// TwinCAT 3 PLC project FB_RobotArm
// Company: DVKruglov
// ProjectVersion: 1.0
// ProgramVersion: 3.1.4023.0
// libraries:
//   Tc2_Standard, * (Beckhoff Automation GmbH)
//   Tc2_System, * (Beckhoff Automation GmbH)
//   Tc3_Module, * (Beckhoff Automation GmbH)
// project tree:
//   FB_RobotArmBase/Constants/ GVL_RobotArmConstants.TcGVL
//   FB_RobotArmBase/Enumeration/ E_RobotArmJointDirection.TcDUT
//   FB_RobotArmBase/ FB_RobotArm.TcPOU
//   FB_RobotArmBase/Structures/ ST_Inputs.TcDUT, ST_Configuration.TcDUT, ST_JointDirection.TcDUT, ST_Outputs.TcDUT
//   FB_RobotArmPickAndPlace/Constants/ GVL_RobotArmPickAndPlaceConstants.TcGVL
//   FB_RobotArmPickAndPlace/Enumeration/ E_BoxPlaceDirection.TcDUT, E_PickPlaceStep.TcDUT
//   FB_RobotArmPickAndPlace/ FB_RobotArmPickAndPlace.TcPOU
//   FB_RobotArmPickAndPlace/Structures/ ST_PickPlaceArmConfig.TcDUT, ST_Places_Inputs.TcDUT
//   / PlcTask.TcTTO (not stored)
//   POUs/ MAIN.TcPOU
// real-time tasks:
//   TASK PlcTask: cycle T#10ms, priority 20, ADS port 350

// ---- FB_RobotArmBase/Enumeration/E_RobotArmJointDirection.TcDUT
{attribute 'qualified_only'}
{attribute 'strict'}
TYPE E_RobotArmJointDirection :
(
	LEFT		:=	1,
	RIGHT		:=	2
);
END_TYPE

// ---- FB_RobotArmBase/Structures/ST_Inputs.TcDUT
TYPE ST_Inputs :
STRUCT
	GRIP_CLOSED    			: BOOL;
	JOINT_FEEDBACK_SIGNAL	: ARRAY [1..GVL_RobotArmConstants.MAX_NUMBER_OF_JOINTS] OF ST_JointDirection;
END_STRUCT
END_TYPE

// ---- FB_RobotArmBase/Structures/ST_Configuration.TcDUT
TYPE ST_Configuration :
STRUCT
	NUMBER_OF_JOINTS	: INT;
END_STRUCT
END_TYPE

// ---- FB_RobotArmBase/Structures/ST_JointDirection.TcDUT
TYPE ST_JointDirection :
STRUCT	
	Left 	: BOOL;
	Right	: BOOL;
END_STRUCT
END_TYPE

// ---- FB_RobotArmBase/Structures/ST_Outputs.TcDUT
TYPE ST_Outputs :
STRUCT	
	GRIP_CLOSE				: BOOL;
	JOINT_TURN		  		: ARRAY [1..GVL_RobotArmConstants.MAX_NUMBER_OF_JOINTS] OF ST_JointDirection; 
END_STRUCT
END_TYPE

// ---- FB_RobotArmPickAndPlace/Enumeration/E_BoxPlaceDirection.TcDUT
{attribute 'qualified_only'}
{attribute 'strict'}
TYPE E_BoxPlaceDirection :
(
	UNDEFINED		:=  0,
	PLACE1_LEFT		:=	1,
	PLACE2_RIGHT	:=	2,
	
	LastPlace
);
END_TYPE

// ---- FB_RobotArmPickAndPlace/Enumeration/E_PickPlaceStep.TcDUT
{attribute 'qualified_only'}
{attribute 'strict'}
TYPE E_PickPlaceStep :
(
	DO_NOTHING 	:= 0,
	MOVE_HAND 	:= 1,
	CHECK_GRIP	:= 2,
	USE_GRIP	:= 3
);
END_TYPE

// ---- FB_RobotArmPickAndPlace/Structures/ST_PickPlaceArmConfig.TcDUT
TYPE ST_PickPlaceArmConfig :
STRUCT

END_STRUCT
END_TYPE

// ---- FB_RobotArmPickAndPlace/Structures/ST_Places_Inputs.TcDUT
TYPE ST_Places_Inputs :
STRUCT
END_STRUCT
END_TYPE

// ---- FB_RobotArmBase/Constants/GVL_RobotArmConstants.TcGVL
{attribute 'qualified_only'}
VAR_GLOBAL CONSTANT
	MAX_NUMBER_OF_JOINTS : INT := 10; // 32 bit => max number is 2^32 - 1
END_VAR

// ---- FB_RobotArmPickAndPlace/Constants/GVL_RobotArmPickAndPlaceConstants.TcGVL
{attribute 'qualified_only'}
VAR_GLOBAL
END_VAR

// ---- FB_RobotArmBase/FB_RobotArm.TcPOU
FUNCTION_BLOCK FB_RobotArm
VAR
	Inputs 		AT%I* 	: ST_Inputs;
	Outputs 	AT%Q* 	: ST_Outputs;
	BaseConfiguration	: ST_Configuration; //REFERENCE TO
	RobotArmJoints 		: ARRAY [1..BaseConfiguration.NUMBER_OF_JOINTS] OF INT;
	Index 				: INT;
	//Joint				: INT := BaseConfiguration.NUMBER_OF_JOINTS;
	InputsDecoupled		: ST_Inputs; 
END_VAR

VAR PERSISTENT
	FirstScan 			: BOOL := TRUE;	
	JointTurnStep		: INT;
END_VAR

_M_StatusUpdate();

METHOD PRIVATE _M_CheckDefaultPosition : BOOL
_M_CheckDefaultPosition := TRUE;

FOR Index := 1 TO BaseConfiguration.NUMBER_OF_JOINTS DO // WHy don't we have if here ???
	_M_CheckDefaultPosition := _M_CheckDefaultPosition AND (NOT InputsDecoupled.JOINT_FEEDBACK_SIGNAL[Index].Right) AND (NOT InputsDecoupled.JOINT_FEEDBACK_SIGNAL[Index].Left);
END_FOR
END_METHOD

METHOD PRIVATE _M_StatusUpdate : BOOL
VAR_INPUT
END_VAR
InputsDecoupled.GRIP_CLOSED := Inputs.GRIP_CLOSED; 

FOR Index := 1 TO BaseConfiguration.NUMBER_OF_JOINTS DO
	InputsDecoupled.JOINT_FEEDBACK_SIGNAL[Index]	:= Inputs.JOINT_FEEDBACK_SIGNAL[Index];
END_FOR
END_METHOD

METHOD PUBLIC M_DefaultPosition : BOOL
M_GripControl( Close := TRUE ); // METHOD( INPUT := , OUTPUT => )
	
FOR Index := 1 TO BaseConfiguration.NUMBER_OF_JOINTS DO 
//	Outputs.JOINT_TURN[Index].Left	:=	FALSE;
//	Outputs.JOINT_TURN[Index].Right	:=	FALSE;
	M_StraightJoint( Joint := Index );
END_FOR
END_METHOD

METHOD PUBLIC M_ForwardKinematics : BOOL
VAR_IN_OUT
	ForwardKinematicsJointControl	: ARRAY[1..GVL_RobotArmConstants.MAX_NUMBER_OF_JOINTS] OF ST_JointDirection; 
END_VAR
// hint: use BaseConfiguration.NUMBER_OF_JOINTS
END_METHOD

METHOD PUBLIC M_GripControl : BOOL
VAR_INPUT
	Close	: BOOL;
END_VAR
Outputs.GRIP_CLOSE := Close;
END_METHOD

METHOD PUBLIC M_StraightJoint : BOOL
VAR_INPUT
	Joint : INT;
END_VAR
Outputs.JOINT_TURN[Joint].Left	:= FALSE;
Outputs.JOINT_TURN[Joint].Right := FALSE;
END_METHOD

METHOD PUBLIC M_TurnJoint
VAR_INPUT
	TurnDirection : INT; // 1 - LEFT, 2 - RIGHT
	
	Joint : INT;
END_VAR
CASE TurnDirection OF 
	E_RobotArmJointDirection.LEFT: // turn left  
		Outputs.JOINT_TURN[Joint].Left	:= TRUE;
	E_RobotArmJointDirection.RIGHT: // turn right
		Outputs.JOINT_TURN[Joint].Right := TRUE;
END_CASE
END_METHOD

PROPERTY PUBLIC P_RobotArmBaseConfiguration : REFERENCE TO ST_Configuration

///Why do we create that properties?
GET
P_RobotArmBaseConfiguration REF= BaseConfiguration;
END_GET
SET
BaseConfiguration REF= P_RobotArmBaseConfiguration;
END_SET
END_PROPERTY

END_FUNCTION_BLOCK

// ---- FB_RobotArmPickAndPlace/FB_RobotArmPickAndPlace.TcPOU
FUNCTION_BLOCK FB_RobotArmPickAndPlace EXTENDS FB_RobotArm
VAR
	
END_VAR

SUPER^();

METHOD PUBLIC M_PickUpFromPlace : BOOL
VAR_INPUT
	PLACE_NUM 	: INT;
END_VAR

VAR_INST
	Step		: INT := 0;
END_VAR
CASE PLACE_NUM OF
	E_BoxPlaceDirection.PLACE1_LEFT: //IF  place1 NOT empty
		Step := E_PickPlaceStep.MOVE_HAND;
		CASE Step OF
			E_PickPlaceStep.DO_NOTHING:
				// do nothing
			E_PickPlaceStep.MOVE_HAND:
				FOR Index := 1 TO BaseConfiguration.NUMBER_OF_JOINTS BY 1 DO
					M_TurnJoint( TurnDirection := E_RobotArmJointDirection.LEFT, Joint := Index);
					
					IF NOT InputsDecoupled.JOINT_LEFT_SIGNAL[Index] THEN
						Index := Index - 1;
					END_IF
				END_FOR
				
				Step := E_PickPlaceStep.CHECK_GRIP;
			
			E_PickPlaceStep.CHECK_GRIP:
				IF InputsDecoupled.GRIP_CLOSED THEN
					Outputs.GRIP_CLOSE := FALSE;
				ELSE
					Step := E_PickPlaceStep.USE_GRIP;
				END_IF
				
			E_PickPlaceStep.USE_GRIP:
				IF NOT InputsDecoupled.GRIP_CLOSED THEN
					Outputs.GRIP_CLOSE := TRUE;
					Step := E_PickPlaceStep.DO_NOTHING;
					PLACE_NUM := E_BoxPlaceDirection.UNDEFINED;
				END_IF
				
		END_CASE
	
	E_BoxPlaceDirection.PLACE2_RIGHT: // //IF  place2 empty
		
	
END_CASE
END_METHOD

METHOD PUBLIC M_PlaceTo : BOOL
VAR_INPUT
	PLACE_NUM : INT;
END_VAR
END_METHOD

END_FUNCTION_BLOCK

// ---- POUs/MAIN.TcPOU
